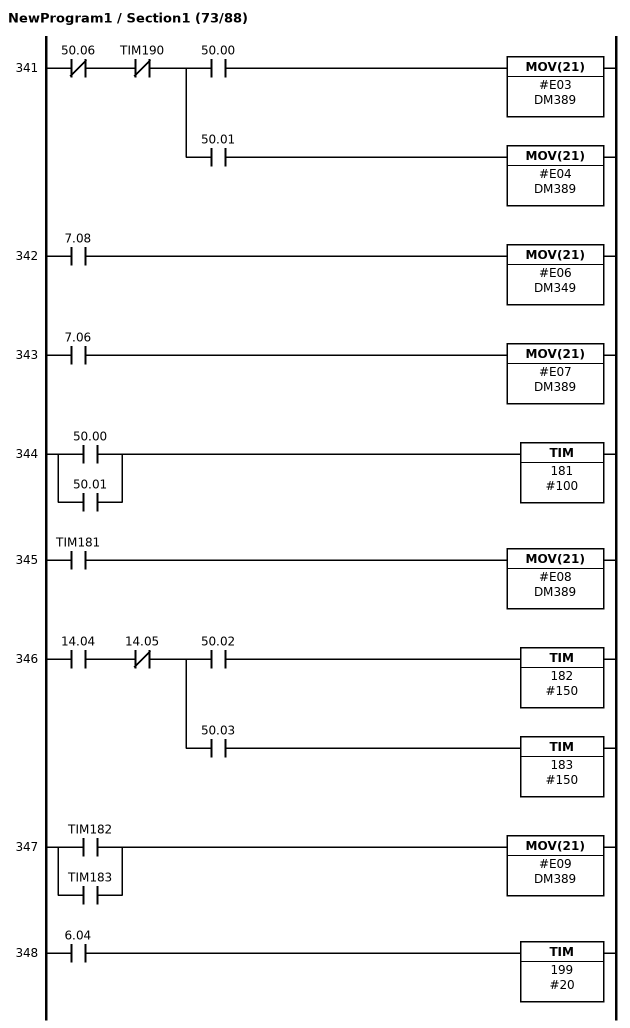
; [picture p72: NewProgram1 / Section1, rungs 341-348]
; rung 341
LDNOT 50.06
ANDNOT TIM190
OUT TR0
AND 50.00
MOV(21) #E03 DM389
LD TR0
AND 50.01
MOV(21) #E04 DM389
; rung 342
LD 7.08
MOV(21) #E06 DM349
; rung 343
LD 7.06
MOV(21) #E07 DM389
; rung 344
LD 50.00
OR 50.01
TIM 181 #100
; rung 345
LD TIM181
MOV(21) #E08 DM389
; rung 346
LD 14.04
ANDNOT 14.05
OUT TR0
AND 50.02
TIM 182 #150
LD TR0
AND 50.03
TIM 183 #150
; rung 347
LD TIM182
OR TIM183
MOV(21) #E09 DM389
; rung 348
LD 6.04
TIM 199 #20

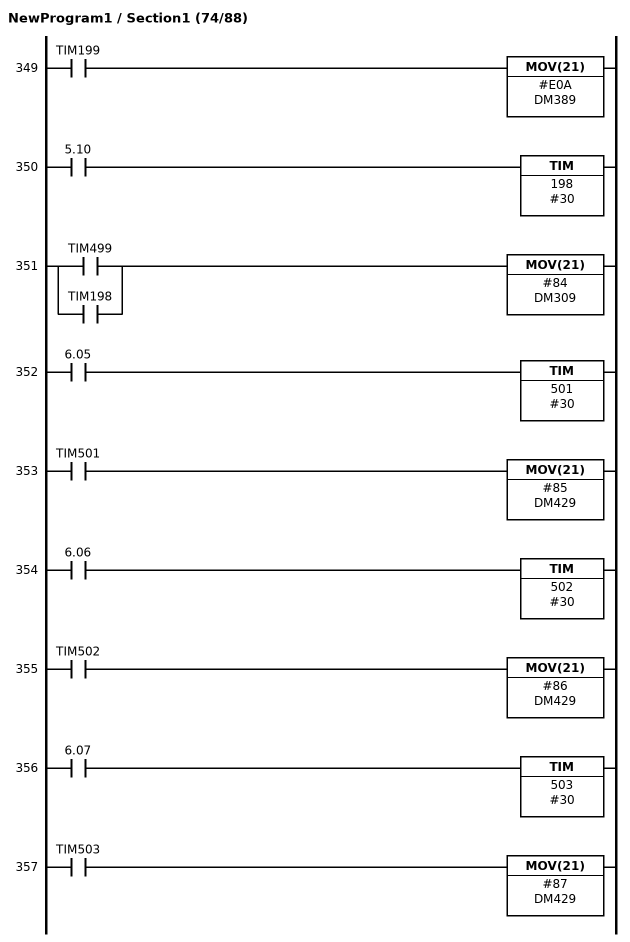
; rung 349
LD TIM199
MOV(21) #E0A DM389
; rung 350
LD 5.10
TIM 198 #30
; rung 351
LD TIM499
OR TIM198
MOV(21) #84 DM309
; rung 352
LD 6.05
TIM 501 #30
; rung 353
LD TIM501
MOV(21) #85 DM429
; rung 354
LD 6.06
TIM 502 #30
; rung 355
LD TIM502
MOV(21) #86 DM429
; rung 356
LD 6.07
TIM 503 #30
; rung 357
LD TIM503
MOV(21) #87 DM429

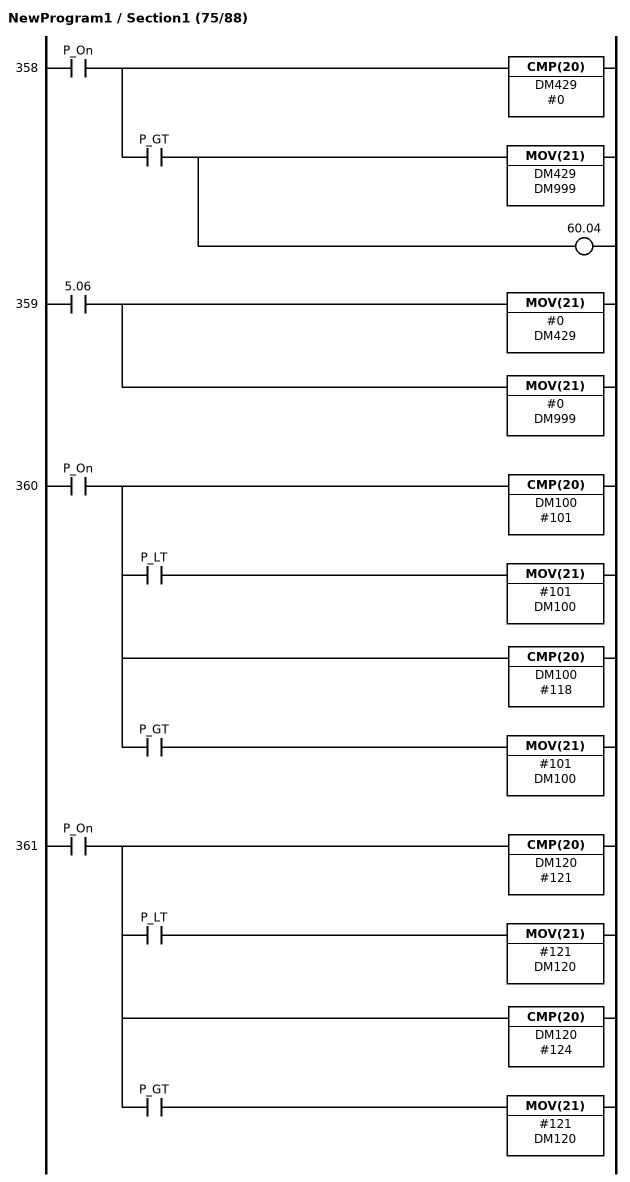
; rung 358
LD P_On
CMP(20) DM429 #0
AND P_GT
MOV(21) DM429 DM999
OUT 60.04
; rung 359
LD 5.06
MOV(21) #0 DM429
MOV(21) #0 DM999
; rung 360
LD P_On
OUT TR0
CMP(20) DM100 #101
AND P_LT
MOV(21) #101 DM100
LD TR0
CMP(20) DM100 #118
AND P_GT
MOV(21) #101 DM100
; rung 361
LD P_On
OUT TR0
CMP(20) DM120 #121
AND P_LT
MOV(21) #121 DM120
LD TR0
CMP(20) DM120 #124
AND P_GT
MOV(21) #121 DM120

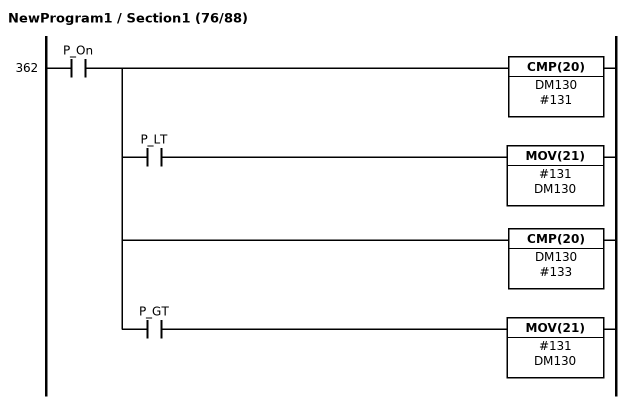
; rung 362
LD P_On
OUT TR0
CMP(20) DM130 #131
AND P_LT
MOV(21) #131 DM130
LD TR0
CMP(20) DM130 #133
AND P_GT
MOV(21) #131 DM130

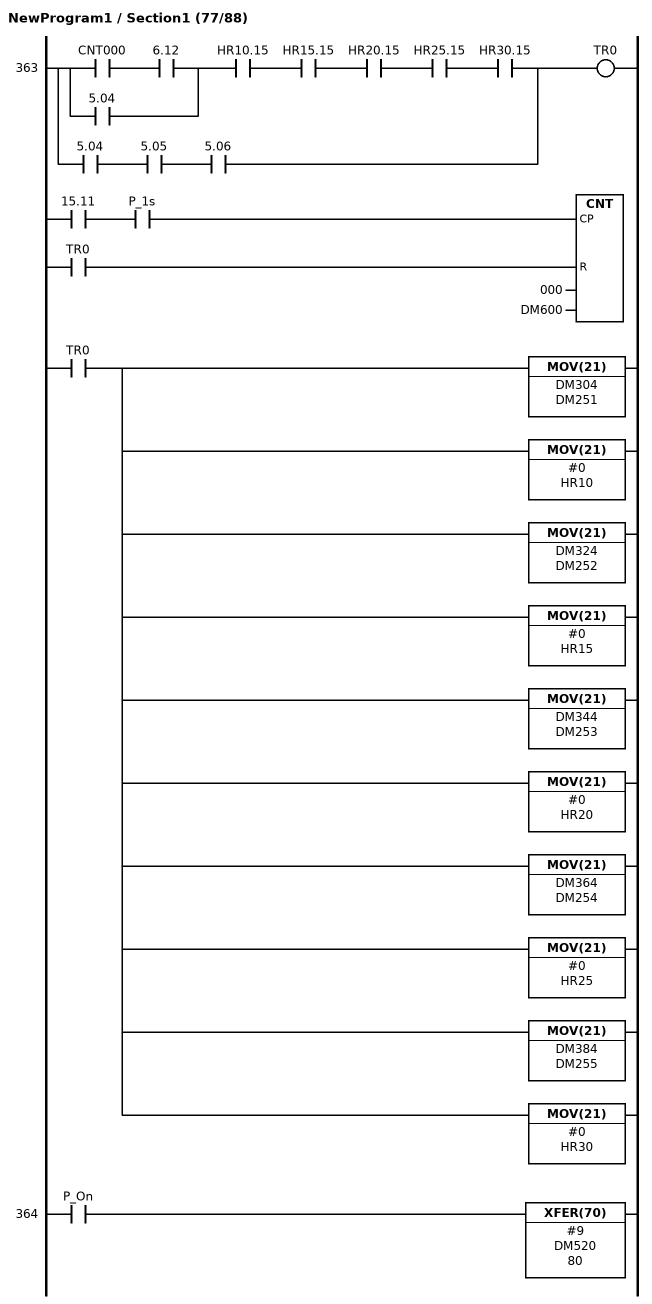
; rung 363
LD 15.11
AND P_1s
LD CNT000
AND 6.12
OR 5.04
AND HR10.15
AND HR15.15
AND HR20.15
AND HR25.15
AND HR30.15
LD 5.04
AND 5.05
AND 5.06
ORLD
OUT TR0
CNT 000 DM600
LD TR0
MOV(21) DM304 DM251
MOV(21) #0 HR10
MOV(21) DM324 DM252
MOV(21) #0 HR15
MOV(21) DM344 DM253
MOV(21) #0 HR20
MOV(21) DM364 DM254
MOV(21) #0 HR25
MOV(21) DM384 DM255
MOV(21) #0 HR30
; rung 364
LD P_On
XFER(70) #9 DM520 80

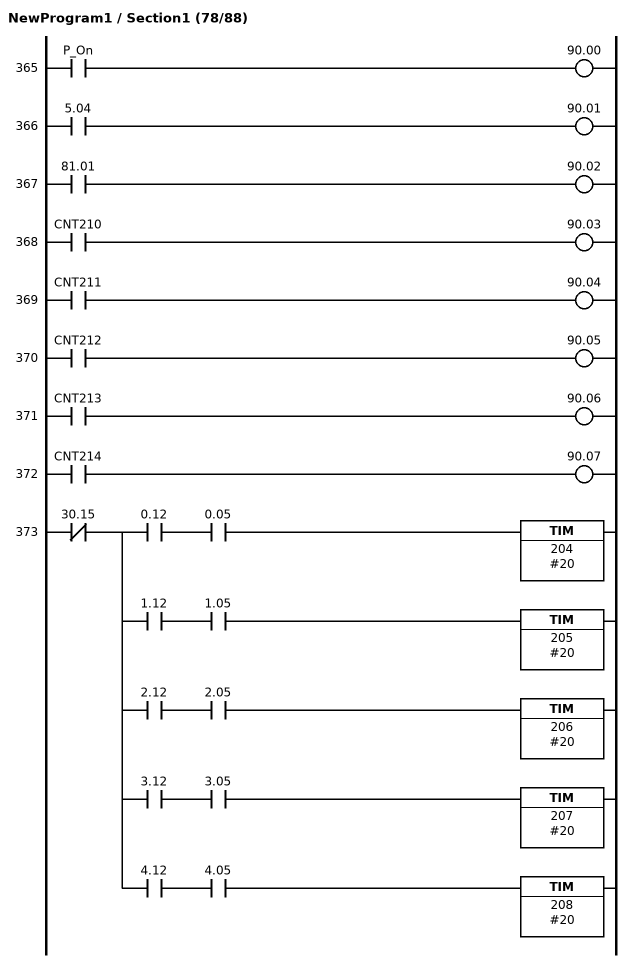
; rung 365
LD P_On
OUT 90.00
; rung 366
LD 5.04
OUT 90.01
; rung 367
LD 81.01
OUT 90.02
; rung 368
LD CNT210
OUT 90.03
; rung 369
LD CNT211
OUT 90.04
; rung 370
LD CNT212
OUT 90.05
; rung 371
LD CNT213
OUT 90.06
; rung 372
LD CNT214
OUT 90.07
; rung 373
LDNOT 30.15
OUT TR0
AND 0.12
AND 0.05
TIM 204 #20
LD TR0
AND 1.12
AND 1.05
TIM 205 #20
LD TR0
AND 2.12
AND 2.05
TIM 206 #20
LD TR0
AND 3.12
AND 3.05
TIM 207 #20
LD TR0
AND 4.12
AND 4.05
TIM 208 #20

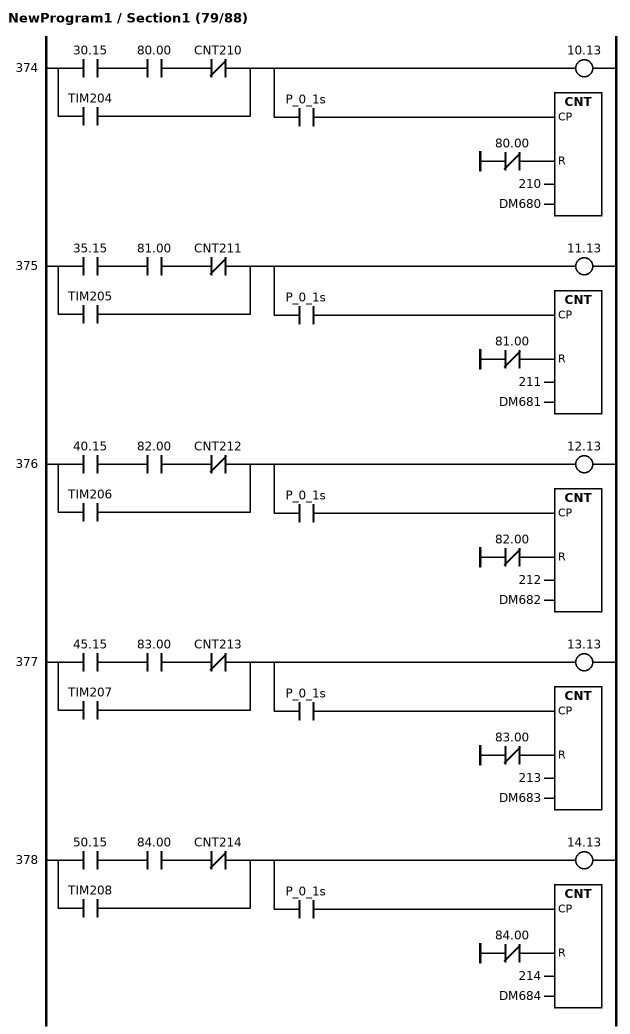
; rung 374
LD 30.15
AND 80.00
ANDNOT CNT210
OR TIM204
OUT 10.13
AND P_0_1s
LDNOT 80.00
CNT 210 DM680
; rung 375
LD 35.15
AND 81.00
ANDNOT CNT211
OR TIM205
OUT 11.13
AND P_0_1s
LDNOT 81.00
CNT 211 DM681
; rung 376
LD 40.15
AND 82.00
ANDNOT CNT212
OR TIM206
OUT 12.13
AND P_0_1s
LDNOT 82.00
CNT 212 DM682
; rung 377
LD 45.15
AND 83.00
ANDNOT CNT213
OR TIM207
OUT 13.13
AND P_0_1s
LDNOT 83.00
CNT 213 DM683
; rung 378
LD 50.15
AND 84.00
ANDNOT CNT214
OR TIM208
OUT 14.13
AND P_0_1s
LDNOT 84.00
CNT 214 DM684

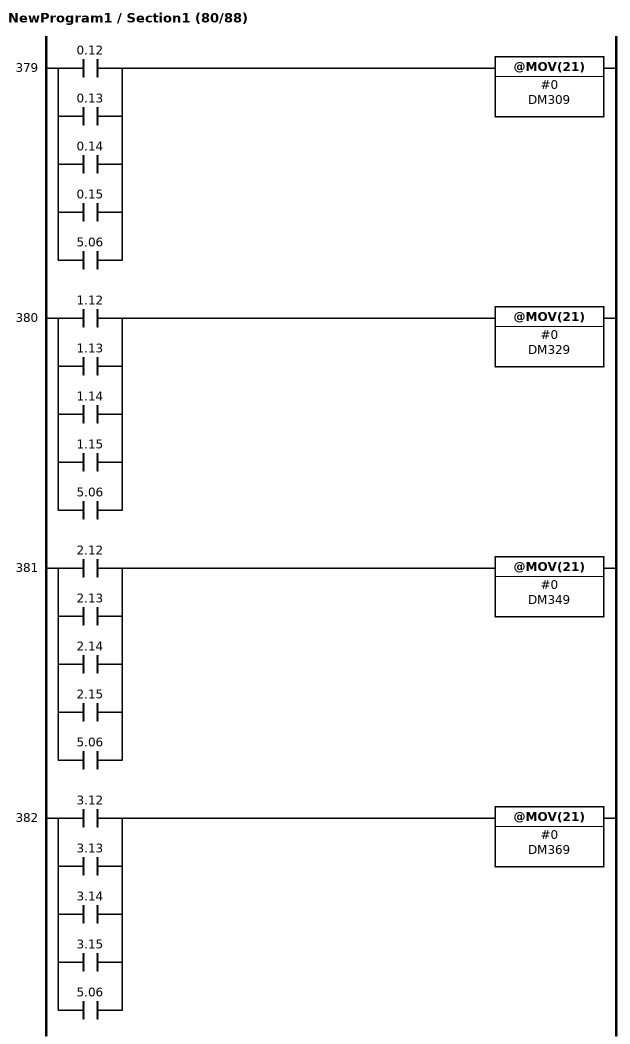
; rung 379
LD 0.12
OR 0.13
OR 0.14
OR 0.15
OR 5.06
@MOV(21) #0 DM309
; rung 380
LD 1.12
OR 1.13
OR 1.14
OR 1.15
OR 5.06
@MOV(21) #0 DM329
; rung 381
LD 2.12
OR 2.13
OR 2.14
OR 2.15
OR 5.06
@MOV(21) #0 DM349
; rung 382
LD 3.12
OR 3.13
OR 3.14
OR 3.15
OR 5.06
@MOV(21) #0 DM369

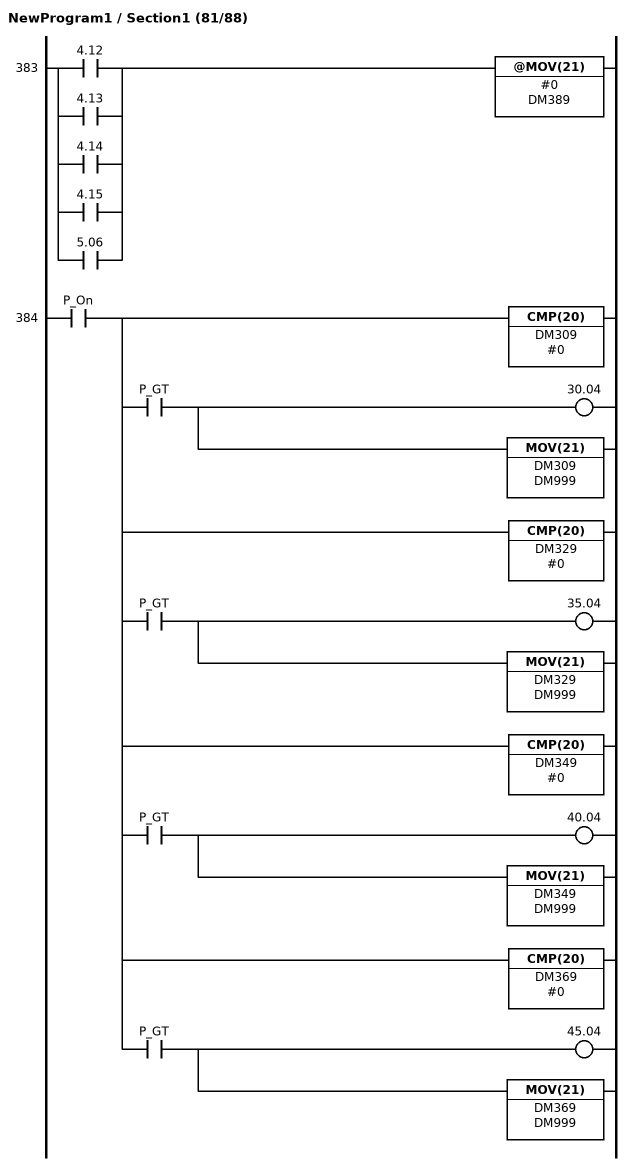
; rung 383
LD 4.12
OR 4.13
OR 4.14
OR 4.15
OR 5.06
@MOV(21) #0 DM389
; rung 384
LD P_On
OUT TR0
CMP(20) DM309 #0
AND P_GT
OUT 30.04
MOV(21) DM309 DM999
LD TR0
CMP(20) DM329 #0
AND P_GT
OUT 35.04
MOV(21) DM329 DM999
LD TR0
CMP(20) DM349 #0
AND P_GT
OUT 40.04
MOV(21) DM349 DM999
LD TR0
CMP(20) DM369 #0
AND P_GT
OUT 45.04
MOV(21) DM369 DM999

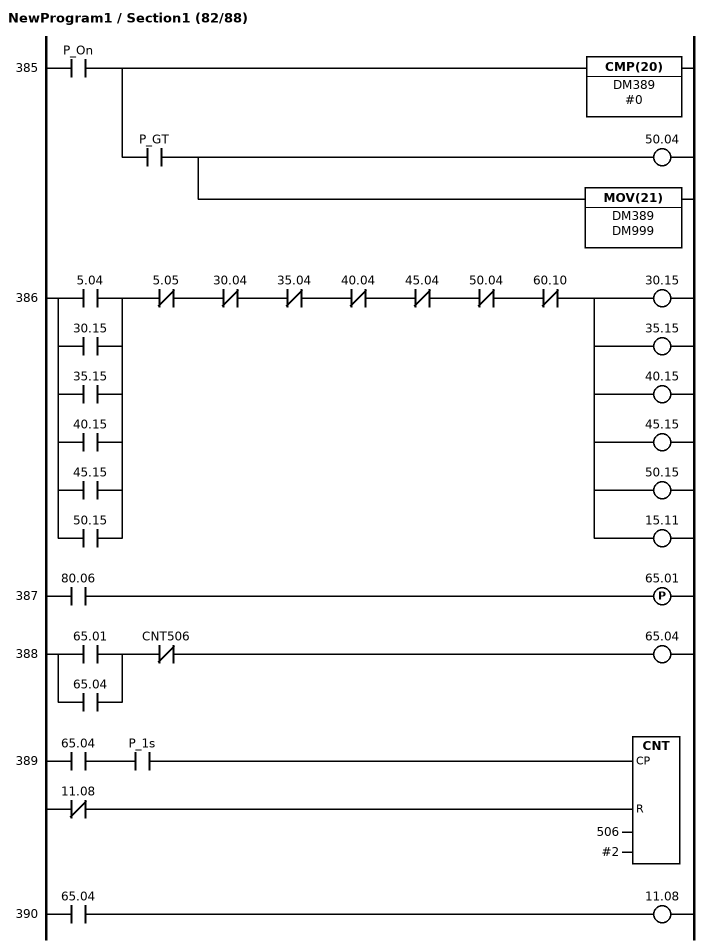
; rung 385
LD P_On
CMP(20) DM389 #0
AND P_GT
OUT 50.04
MOV(21) DM389 DM999
; rung 386
LD 5.04
OR 30.15
OR 35.15
OR 40.15
OR 45.15
OR 50.15
ANDNOT 5.05
ANDNOT 30.04
ANDNOT 35.04
ANDNOT 40.04
ANDNOT 45.04
ANDNOT 50.04
ANDNOT 60.10
OUT 30.15
OUT 35.15
OUT 40.15
OUT 45.15
OUT 50.15
OUT 15.11
; rung 387
LD 80.06
DIFU(13) 65.01
; rung 388
LD 65.01
OR 65.04
ANDNOT CNT506
OUT 65.04
; rung 389
LD 65.04
AND P_1s
LDNOT 11.08
CNT 506 #2
; rung 390
LD 65.04
OUT 11.08

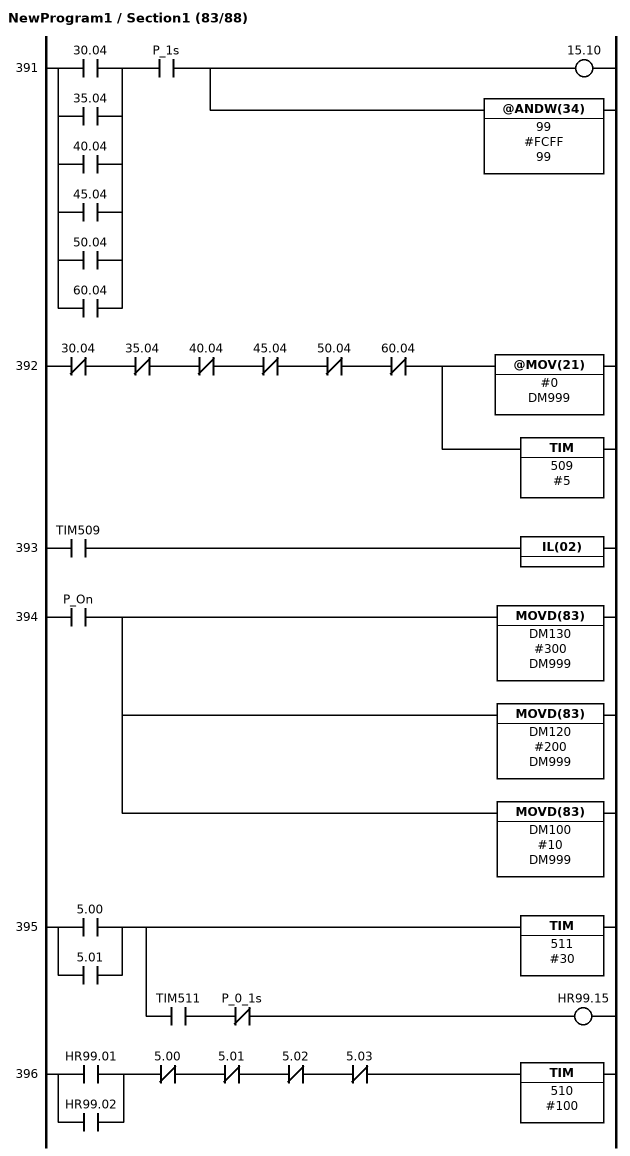
; rung 391
LD 30.04
OR 35.04
OR 40.04
OR 45.04
OR 50.04
OR 60.04
AND P_1s
OUT 15.10
@ANDW(34) 99 #FCFF 99
; rung 392
LDNOT 30.04
ANDNOT 35.04
ANDNOT 40.04
ANDNOT 45.04
ANDNOT 50.04
ANDNOT 60.04
@MOV(21) #0 DM999
TIM 509 #5
; rung 393
LD TIM509
IL(02)
; rung 394
LD P_On
MOVD(83) DM130 #300 DM999
MOVD(83) DM120 #200 DM999
MOVD(83) DM100 #10 DM999
; rung 395
LD 5.00
OR 5.01
TIM 511 #30
AND TIM511
ANDNOT P_0_1s
OUT HR99.15
; rung 396
LD HR99.01
OR HR99.02
ANDNOT 5.00
ANDNOT 5.01
ANDNOT 5.02
ANDNOT 5.03
TIM 510 #100

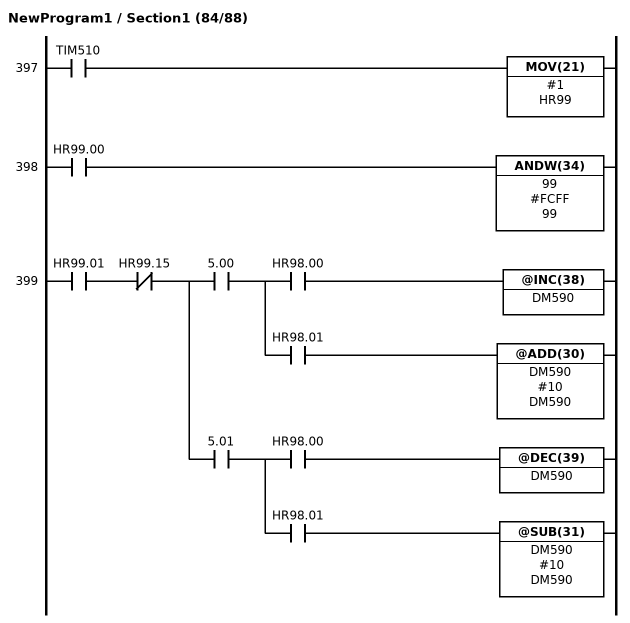
; rung 397
LD TIM510
MOV(21) #1 HR99
; rung 398
LD HR99.00
ANDW(34) 99 #FCFF 99
; rung 399
LD HR99.01
ANDNOT HR99.15
OUT TR0
AND 5.00
OUT TR1
AND HR98.00
@INC(38) DM590
LD TR1
AND HR98.01
@ADD(30) DM590 #10 DM590
LD TR0
AND 5.01
OUT TR0
AND HR98.00
@DEC(39) DM590
LD TR0
AND HR98.01
@SUB(31) DM590 #10 DM590

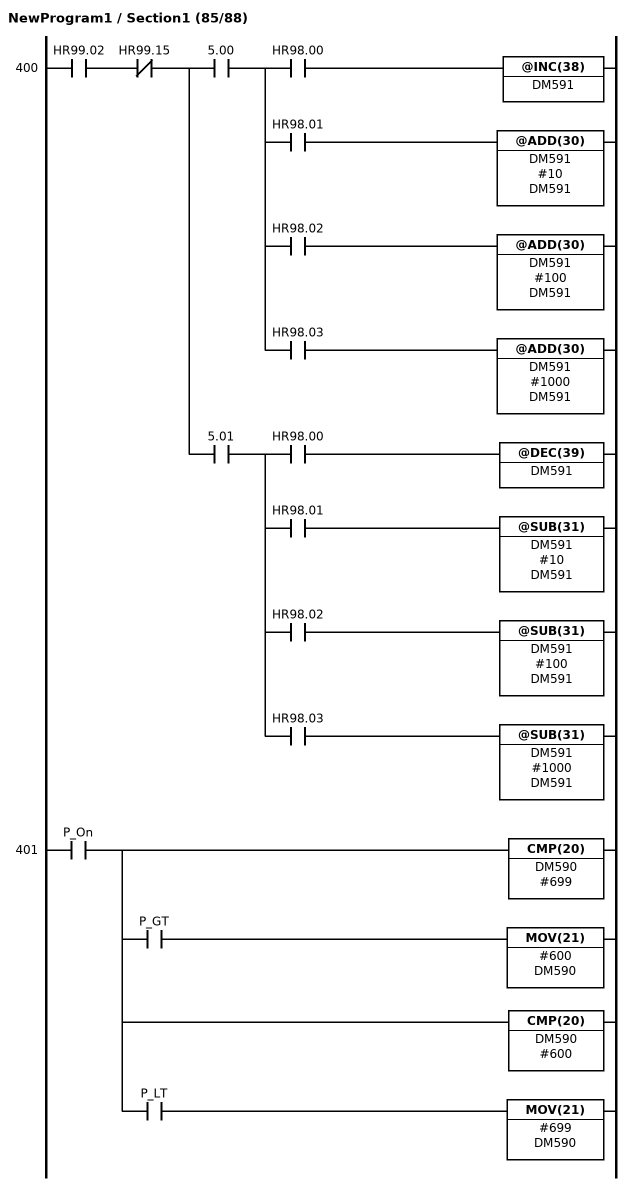
; rung 400
LD HR99.02
ANDNOT HR99.15
OUT TR0
AND 5.00
OUT TR1
AND HR98.00
@INC(38) DM591
LD TR1
AND HR98.01
@ADD(30) DM591 #10 DM591
LD TR1
AND HR98.02
@ADD(30) DM591 #100 DM591
LD TR1
AND HR98.03
@ADD(30) DM591 #1000 DM591
LD TR0
AND 5.01
OUT TR0
AND HR98.00
@DEC(39) DM591
LD TR0
AND HR98.01
@SUB(31) DM591 #10 DM591
LD TR0
AND HR98.02
@SUB(31) DM591 #100 DM591
LD TR0
AND HR98.03
@SUB(31) DM591 #1000 DM591
; rung 401
LD P_On
OUT TR0
CMP(20) DM590 #699
AND P_GT
MOV(21) #600 DM590
LD TR0
CMP(20) DM590 #600
AND P_LT
MOV(21) #699 DM590

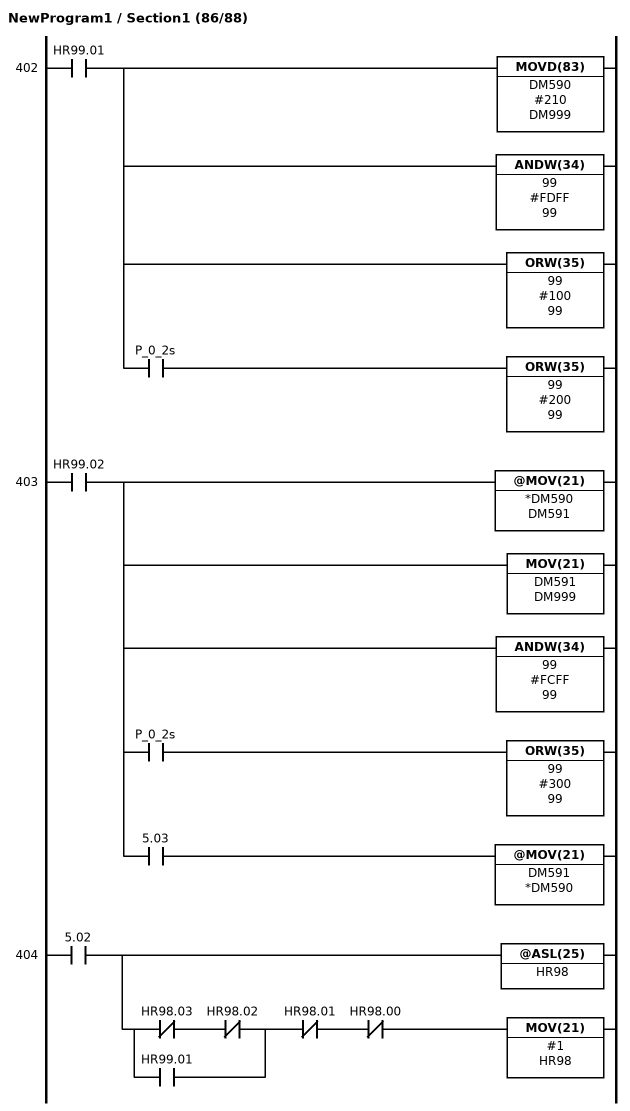
; rung 402
LD HR99.01
MOVD(83) DM590 #210 DM999
ANDW(34) 99 #FDFF 99
ORW(35) 99 #100 99
AND P_0_2s
ORW(35) 99 #200 99
; rung 403
LD HR99.02
OUT TR0
@MOV(21) *DM590 DM591
MOV(21) DM591 DM999
ANDW(34) 99 #FCFF 99
AND P_0_2s
ORW(35) 99 #300 99
LD TR0
AND 5.03
@MOV(21) DM591 *DM590
; rung 404
LD 5.02
@ASL(25) HR98
LDNOT HR98.03
ANDNOT HR98.02
OR HR99.01
ANDLD
ANDNOT HR98.01
ANDNOT HR98.00
MOV(21) #1 HR98

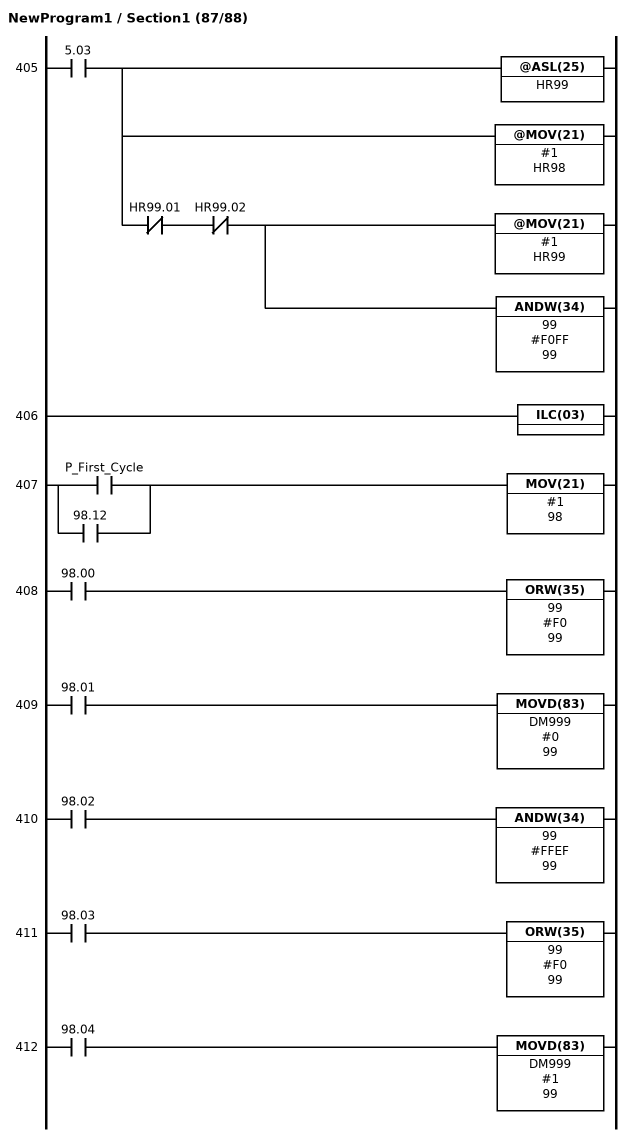
; rung 405
LD 5.03
@ASL(25) HR99
@MOV(21) #1 HR98
ANDNOT HR99.01
ANDNOT HR99.02
@MOV(21) #1 HR99
ANDW(34) 99 #F0FF 99
; rung 406
ILC(03)
; rung 407
LD P_First_Cycle
OR 98.12
MOV(21) #1 98
; rung 408
LD 98.00
ORW(35) 99 #F0 99
; rung 409
LD 98.01
MOVD(83) DM999 #0 99
; rung 410
LD 98.02
ANDW(34) 99 #FFEF 99
; rung 411
LD 98.03
ORW(35) 99 #F0 99
; rung 412
LD 98.04
MOVD(83) DM999 #1 99

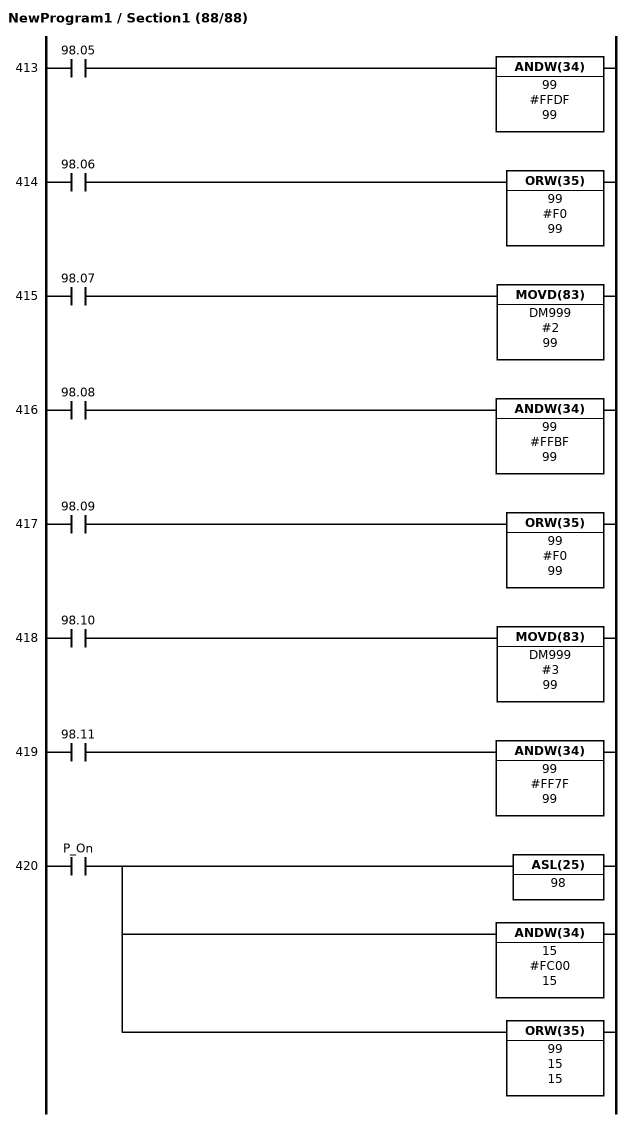
; rung 413
LD 98.05
ANDW(34) 99 #FFDF 99
; rung 414
LD 98.06
ORW(35) 99 #F0 99
; rung 415
LD 98.07
MOVD(83) DM999 #2 99
; rung 416
LD 98.08
ANDW(34) 99 #FFBF 99
; rung 417
LD 98.09
ORW(35) 99 #F0 99
; rung 418
LD 98.10
MOVD(83) DM999 #3 99
; rung 419
LD 98.11
ANDW(34) 99 #FF7F 99
; rung 420
LD P_On
ASL(25) 98
ANDW(34) 15 #FC00 15
ORW(35) 99 15 15
; rung 421
END(01)